// TwinCAT 3 PLC project TcUnit_Tests1
// ProgramVersion: 3.1.4024.0
// libraries:
//   Tc2_Standard, * (Beckhoff Automation GmbH)
//   Tc2_System, * (Beckhoff Automation GmbH)
//   Tc3_Module, * (Beckhoff Automation GmbH)
//   TcUnit, * (www.tcunit.org)
// project tree:
//   / PlcTask.TcTTO
//   POUs/ FB_Add2Ints.TcPOU, FB_Add2Ints_Test.TcPOU, FB_Multiply2Ints.TcPOU, FB_ToMakeSureThePLCWorks.TcPOU, MAIN.TcPOU

CONFIGURATION TcUnit_Tests1
    RESOURCE PLC ON TwinCAT3
        TASK PlcTask(INTERVAL := T#10ms, PRIORITY := 20);
        PROGRAM MAIN WITH PlcTask : MAIN;
    END_RESOURCE
END_CONFIGURATION

// ---- POUs/MAIN.TcPOU
PROGRAM MAIN
VAR
//	fbtest1 : FB_ToMakeSureThePLCWorks;
	fbAdd2Ints_Test : FB_Add2Ints_Test;
END_VAR

TcUnit.RUN();

END_PROGRAM

// ---- POUs/FB_Add2Ints_Test.TcPOU
FUNCTION_BLOCK FB_Add2Ints_Test EXTENDS TcUnit.FB_TestSuite

METHOD PRIVATE Add5Plus10Expect15 
VAR
	fbAdd	: FB_Add2Ints;
	result	: INT;
END_VAR
TEST('Add5Plus10Expect15');
fbAdd(Int1 := 5, Int2 := 10, Result => result);
	
AssertEquals_Int(Expected := 15, Actual := result, Message :='Didnt work');
AssertFalse(Condition := TRUE, Message := 'should fail');	

TEST_FINISHED();
END_METHOD

END_FUNCTION_BLOCK

// ---- POUs/FB_Add2Ints.TcPOU
FUNCTION_BLOCK FB_Add2Ints
VAR_INPUT
	Int1	: INT;
	Int2	: INT;
END_VAR
VAR_OUTPUT
	Result	: INT;
END_VAR
VAR
END_VAR

END_FUNCTION_BLOCK

// ---- POUs/FB_Multiply2Ints.TcPOU
FUNCTION_BLOCK FB_Multiply2Ints
VAR_INPUT
	Int1	: INT;
	Int2	: INT;
END_VAR
VAR_OUTPUT
	Result	: INT;
END_VAR

Result := Int1 * Int2;

END_FUNCTION_BLOCK

// ---- POUs/FB_ToMakeSureThePLCWorks.TcPOU
FUNCTION_BLOCK FB_ToMakeSureThePLCWorks

VAR
	fbMult	: FB_Multiply2Ints;
	result	: INT;
END_VAR

fbMult(Int1 := 2, Int2 := 15, Result => result);

END_FUNCTION_BLOCK
